# EPICS substitutions: iocs/miroTest/miroTestApp/Db/miroCamera.substitutions
file phantomCamera.template {
pattern{ P, R , PORT, ADDR, TIMEOUT}
{ "test:", "ioc:" , "PHANTOM", 0, 1}
}
